(*********************************** G.D S.p.A. - Technical Department ***********************************
============= PROGRAM INFO ============
FOLDER:             TBD
MACHINES INVOLVED:  TBD 

============= DESCRIPTION =============
csp machine declaration

============= REVISIONS ===============
Date		Version	 	Author      	Description             
----------	-------		------------  	--------------------------------------------
2019/04/05 	0000.00	 	M.Grasso		Creation of the PRG

**********************************************************************************************************)
(*$R process_ref := prc; $*)
PROGRAM csp_transfer_infeed_metering
	
VAR
	
	prc:									process;
	prc_path:								STRING;

	disable_req:							BOOL;

END_VAR

_read_var_input();

_object_manager();

IF NOT objects_running()
THEN
	RETURN;	
END_IF

_read_process_image();

_mode_manager();

CASE process_get_mode(prc) OF
	MODE_ABSENT,
	MODE_INACTIVE:
		RETURN;
	MODE_TEST:
		_handle_process_test();
END_CASE


_set_runtime_properties();

(*************************************************************************************
**************************************************************************************)
(*BODY*)

disable_req := NOT
				((
				csp_transfer_infeed.run_infeed_belts
				)
				AND
				process_is_ready(prc)
				AND
				process_subtree_is_ready(prc));
						


(************************************************************************)
(************************************************************************)

_handle_messages();

_write_output();

ACTION _handle_messages:
;
END_ACTION

ACTION _handle_process_test:
;
END_ACTION

ACTION _mode_manager:
IF process_mode_req_is_pending(prc)
THEN
    process_apply_mode_req_first_step(prc);
    CASE process_get_mode(prc) OF
        MODE_TO_ABSENT:
			;
        MODE_TO_INACTIVE:
			;
        MODE_TO_TEST:
			;
        MODE_TO_OPERATIONAL:
			;
    END_CASE
    process_apply_mode_req_second_step(prc);
END_IF
END_ACTION

ACTION _object_manager:
IF objects_initialization()
THEN
	sub_process_init(
		object_name					:= 'csp_transfer_infeed_metering.prc', 
		process						:= csp_transfer_infeed.prc, 
		CONVERSION_this				:= prc);
		
	prc_path 						:= process_get_path(prc);
	

END_IF

IF objects_running()
THEN
	process_cycle(prc);
END_IF
END_ACTION

ACTION _read_process_image:
;
END_ACTION

ACTION _read_var_input:
;
END_ACTION

ACTION _set_runtime_properties:
;
END_ACTION

ACTION _write_output:
;
END_ACTION

END_PROGRAM

(* stored: Version 1.1.0.1, ProductVersion 3.1.4024.3
   POU csp_transfer_infeed_metering: Id {5a9db858-609e-4d22-8669-1534abf60dfd}, SpecialFunc None
   Action _handle_messages: Id {ef33c87c-55b6-4a2a-9027-6dcdc31d22ce}
   Action _handle_process_test: Id {f0027c4a-582b-4f06-a168-b3d466f0ebbc}
   Action _mode_manager: Id {a71b5a8a-fbe6-421c-b090-72577e591ceb}
   Action _object_manager: Id {61a94ebc-7316-4a8a-ac0d-24967ff537e9}
   Action _read_process_image: Id {8763950d-7825-4cd8-a823-dc3c6dfecf2f}
   Action _read_var_input: Id {7e67c105-b7eb-4ec9-adf9-fe8202cd9675}
   Action _set_runtime_properties: Id {504c4c29-ddb3-4e64-89aa-9669af6b3980}
   Action _write_output: Id {fa9bd4f6-8d9f-43d3-a47b-c00a4a906842} *)
